SYSTEM AgSYS (* System Configuration *)
  (* Standard: 61499-1 *)
  (* Version 1.0, 2010-04-25, Unknown, TUT *)
  APPLICATION APP1
  END_APPLICATION
  DEVICE HMI : FRAME_DEVICE(BOUNDS := [200,0,800,450], GRID := [3,4])
    RESOURCE HMIPanelMain : PANEL_RESOURCE
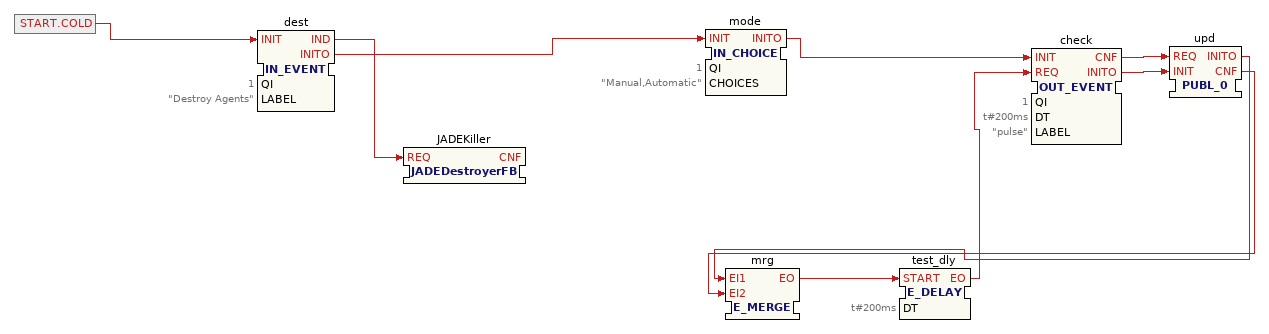
      FBS
        dest : IN_EVENT(QI := 1, LABEL := "Destroy Agents");
        JADEKiller : JADEDestroyerFB;
        mode : IN_CHOICE(QI := 1, CHOICES := "Manual,Automatic");
        check : OUT_EVENT(QI := 1, DT := t#200ms, LABEL := "pulse");
        test_dly : E_DELAY(DT := t#200ms);
        upd : PUBL_0;
        mrg : E_MERGE;
      END_FBS
      EVENT_CONNECTIONS
        START.COLD TO dest.INIT;
        dest.IND TO JADEKiller.REQ;
        dest.INITO TO mode.INIT;
        mode.INITO TO check.INIT;
        test_dly.EO TO check.REQ;
        check.CNF TO upd.REQ;
        upd.INITO TO mrg.EI1;
        upd.CNF TO mrg.EI2;
        mrg.EO TO test_dly.START;
        check.INITO TO upd.INIT;
      END_CONNECTIONS
    END_RESOURCE
    RESOURCE WS2 : PANEL_RESOURCE(ROWS := 4, COLS := 2)
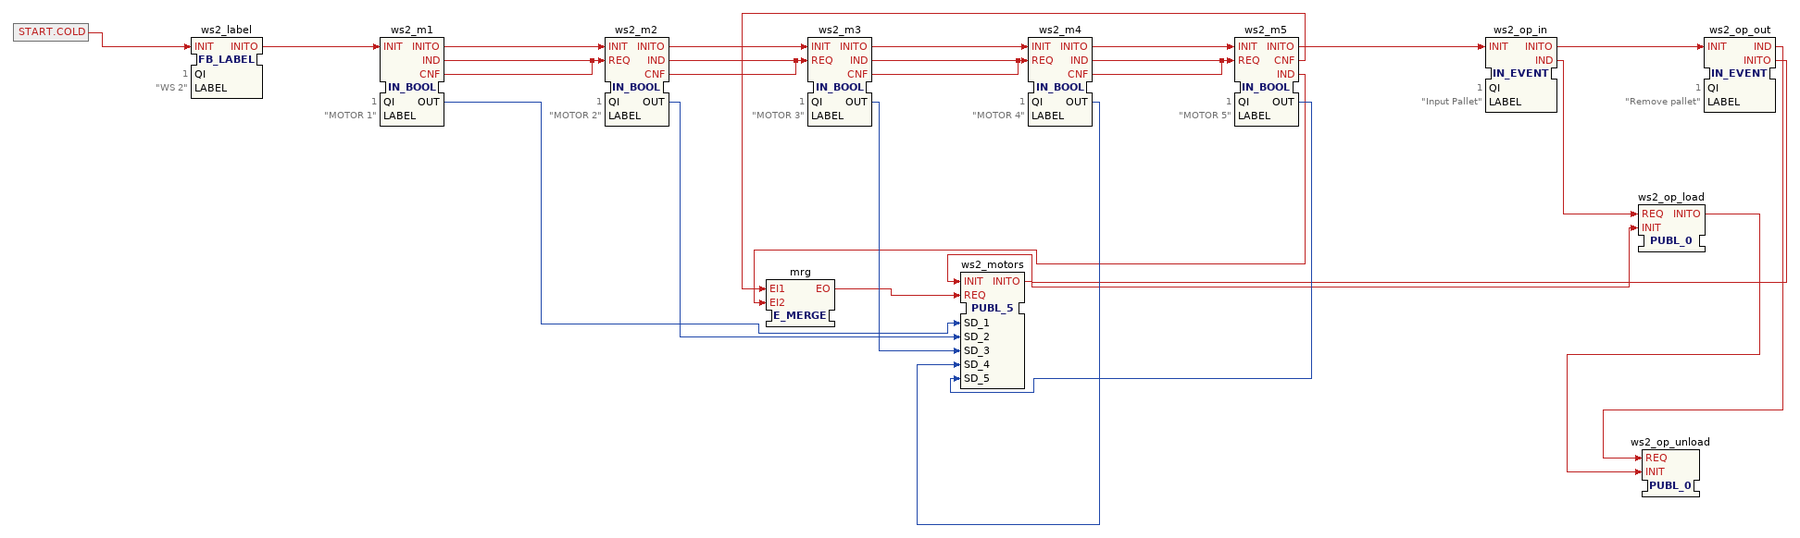
      FBS
        ws2_label : FB_LABEL(QI := 1, LABEL := "WS 2");
        ws2_m1 : IN_BOOL(QI := 1, LABEL := "MOTOR 1");
        ws2_m2 : IN_BOOL(QI := 1, LABEL := "MOTOR 2");
        ws2_m3 : IN_BOOL(QI := 1, LABEL := "MOTOR 3");
        ws2_m4 : IN_BOOL(QI := 1, LABEL := "MOTOR 4");
        ws2_m5 : IN_BOOL(QI := 1, LABEL := "MOTOR 5");
        ws2_op_in : IN_EVENT(QI := 1, LABEL := "Input Pallet");
        ws2_op_out : IN_EVENT(QI := 1, LABEL := "Remove pallet");
        ws2_motors : PUBL_5;
        ws2_op_load : PUBL_0;
        ws2_op_unload : PUBL_0;
        mrg : E_MERGE;
      END_FBS
      EVENT_CONNECTIONS
        START.COLD TO ws2_label.INIT;
        ws2_label.INITO TO ws2_m1.INIT;
        ws2_m1.INITO TO ws2_m2.INIT;
        ws2_m2.INITO TO ws2_m3.INIT;
        ws2_m3.INITO TO ws2_m4.INIT;
        ws2_m4.INITO TO ws2_m5.INIT;
        ws2_m5.INITO TO ws2_op_in.INIT;
        ws2_op_in.INITO TO ws2_op_out.INIT;
        ws2_m1.IND TO ws2_m2.REQ;
        ws2_m2.IND TO ws2_m3.REQ;
        ws2_m3.IND TO ws2_m4.REQ;
        ws2_m4.IND TO ws2_m5.REQ;
        ws2_op_in.IND TO ws2_op_load.REQ;
        ws2_op_out.IND TO ws2_op_unload.REQ;
        ws2_op_out.INITO TO ws2_motors.INIT;
        ws2_motors.INITO TO ws2_op_load.INIT;
        ws2_op_load.INITO TO ws2_op_unload.INIT;
        ws2_m5.CNF TO mrg.EI1;
        ws2_m5.IND TO mrg.EI2;
        mrg.EO TO ws2_motors.REQ;
        ws2_m3.CNF TO ws2_m4.REQ;
        ws2_m4.CNF TO ws2_m5.REQ;
        ws2_m2.CNF TO ws2_m3.REQ;
        ws2_m1.CNF TO ws2_m2.REQ;
      END_CONNECTIONS
      DATA_CONNECTIONS
        ws2_m1.OUT TO ws2_motors.SD_1;
        ws2_m2.OUT TO ws2_motors.SD_2;
        ws2_m3.OUT TO ws2_motors.SD_3;
        ws2_m4.OUT TO ws2_motors.SD_4;
        ws2_m5.OUT TO ws2_motors.SD_5;
      END_CONNECTIONS
    END_RESOURCE
    RESOURCE WS4 : PANEL_RESOURCE(ROWS := 4, COLS := 2)
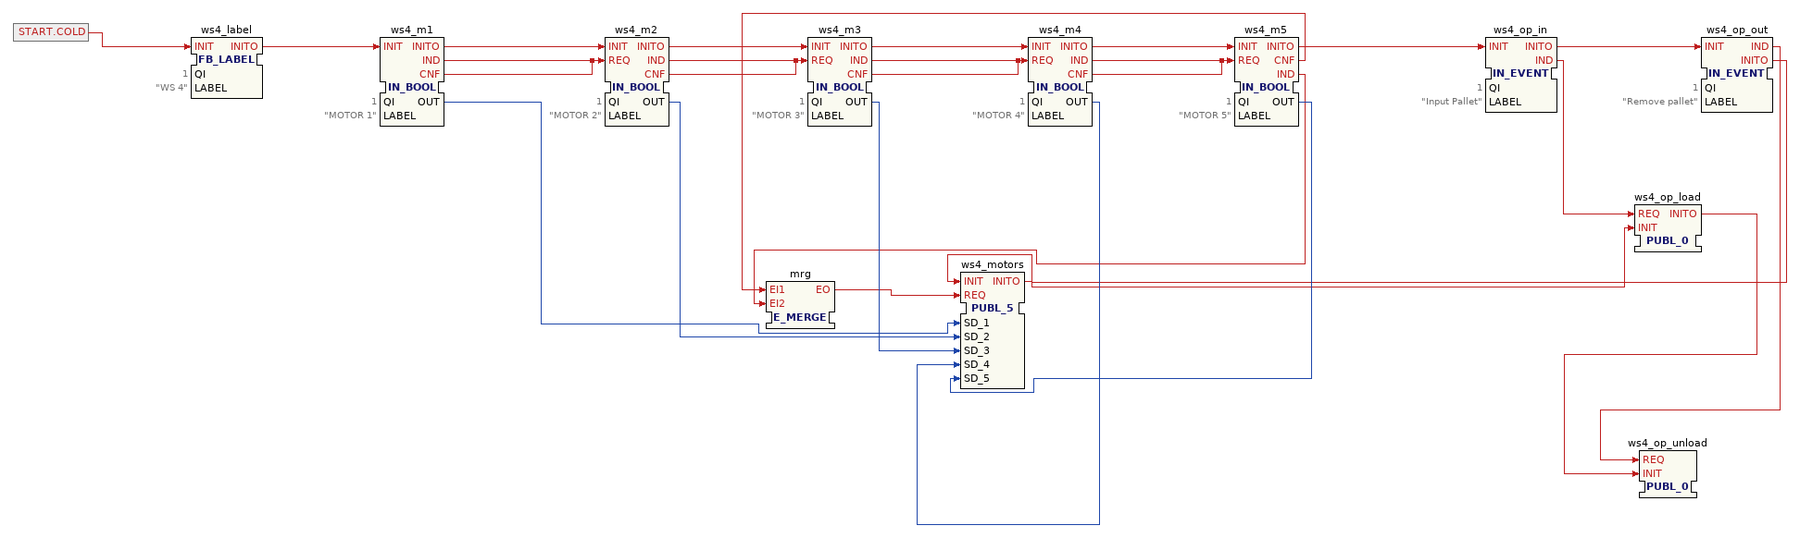
      FBS
        ws4_label : FB_LABEL(QI := 1, LABEL := "WS 4");
        ws4_m1 : IN_BOOL(QI := 1, LABEL := "MOTOR 1");
        ws4_m2 : IN_BOOL(QI := 1, LABEL := "MOTOR 2");
        ws4_m3 : IN_BOOL(QI := 1, LABEL := "MOTOR 3");
        ws4_m4 : IN_BOOL(QI := 1, LABEL := "MOTOR 4");
        ws4_m5 : IN_BOOL(QI := 1, LABEL := "MOTOR 5");
        ws4_op_in : IN_EVENT(QI := 1, LABEL := "Input Pallet");
        ws4_op_out : IN_EVENT(QI := 1, LABEL := "Remove pallet");
        ws4_motors : PUBL_5;
        ws4_op_load : PUBL_0;
        ws4_op_unload : PUBL_0;
        mrg : E_MERGE;
      END_FBS
      EVENT_CONNECTIONS
        START.COLD TO ws4_label.INIT;
        ws4_label.INITO TO ws4_m1.INIT;
        ws4_m1.INITO TO ws4_m2.INIT;
        ws4_m2.INITO TO ws4_m3.INIT;
        ws4_m3.INITO TO ws4_m4.INIT;
        ws4_m4.INITO TO ws4_m5.INIT;
        ws4_m5.INITO TO ws4_op_in.INIT;
        ws4_op_in.INITO TO ws4_op_out.INIT;
        ws4_m1.IND TO ws4_m2.REQ;
        ws4_m2.IND TO ws4_m3.REQ;
        ws4_m3.IND TO ws4_m4.REQ;
        ws4_m4.IND TO ws4_m5.REQ;
        ws4_op_in.IND TO ws4_op_load.REQ;
        ws4_op_out.IND TO ws4_op_unload.REQ;
        ws4_op_out.INITO TO ws4_motors.INIT;
        ws4_motors.INITO TO ws4_op_load.INIT;
        ws4_op_load.INITO TO ws4_op_unload.INIT;
        ws4_m5.CNF TO mrg.EI1;
        ws4_m5.IND TO mrg.EI2;
        mrg.EO TO ws4_motors.REQ;
        ws4_m3.CNF TO ws4_m4.REQ;
        ws4_m4.CNF TO ws4_m5.REQ;
        ws4_m2.CNF TO ws4_m3.REQ;
        ws4_m1.CNF TO ws4_m2.REQ;
      END_CONNECTIONS
      DATA_CONNECTIONS
        ws4_m1.OUT TO ws4_motors.SD_1;
        ws4_m2.OUT TO ws4_motors.SD_2;
        ws4_m3.OUT TO ws4_motors.SD_3;
        ws4_m4.OUT TO ws4_motors.SD_4;
        ws4_m5.OUT TO ws4_motors.SD_5;
      END_CONNECTIONS
    END_RESOURCE
    RESOURCE empt1 : PANEL_RESOURCE
    END_RESOURCE
    RESOURCE Start_Lifter : PANEL_RESOURCE(ROWS := 3, COLS := 1)
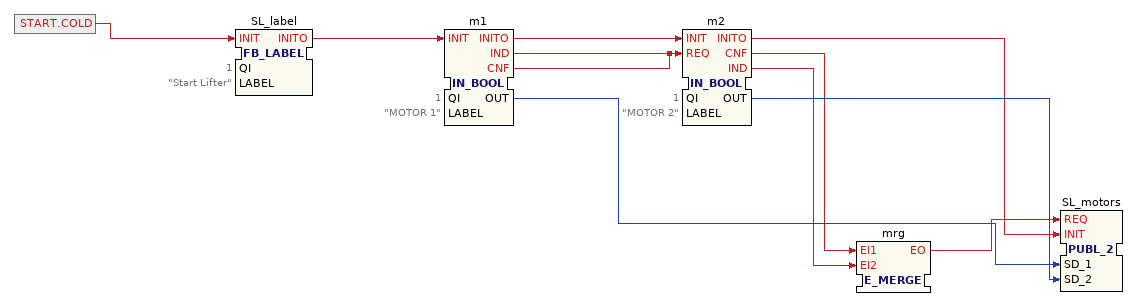
      FBS
        SL_label : FB_LABEL(QI := 1, LABEL := "Start Lifter");
        m1 : IN_BOOL(QI := 1, LABEL := "MOTOR 1");
        m2 : IN_BOOL(QI := 1, LABEL := "MOTOR 2");
        SL_motors : PUBL_2;
        mrg : E_MERGE;
      END_FBS
      EVENT_CONNECTIONS
        START.COLD TO SL_label.INIT;
        m1.INITO TO m2.INIT;
        m1.IND TO m2.REQ;
        mrg.EO TO SL_motors.REQ;
        m1.CNF TO m2.REQ;
        m2.INITO TO SL_motors.INIT;
        m2.CNF TO mrg.EI1;
        m2.IND TO mrg.EI2;
        SL_label.INITO TO m1.INIT;
      END_CONNECTIONS
      DATA_CONNECTIONS
        m1.OUT TO SL_motors.SD_1;
        m2.OUT TO SL_motors.SD_2;
      END_CONNECTIONS
    END_RESOURCE
    RESOURCE ML1 : PANEL_RESOURCE(ROWS := 3, COLS := 2)
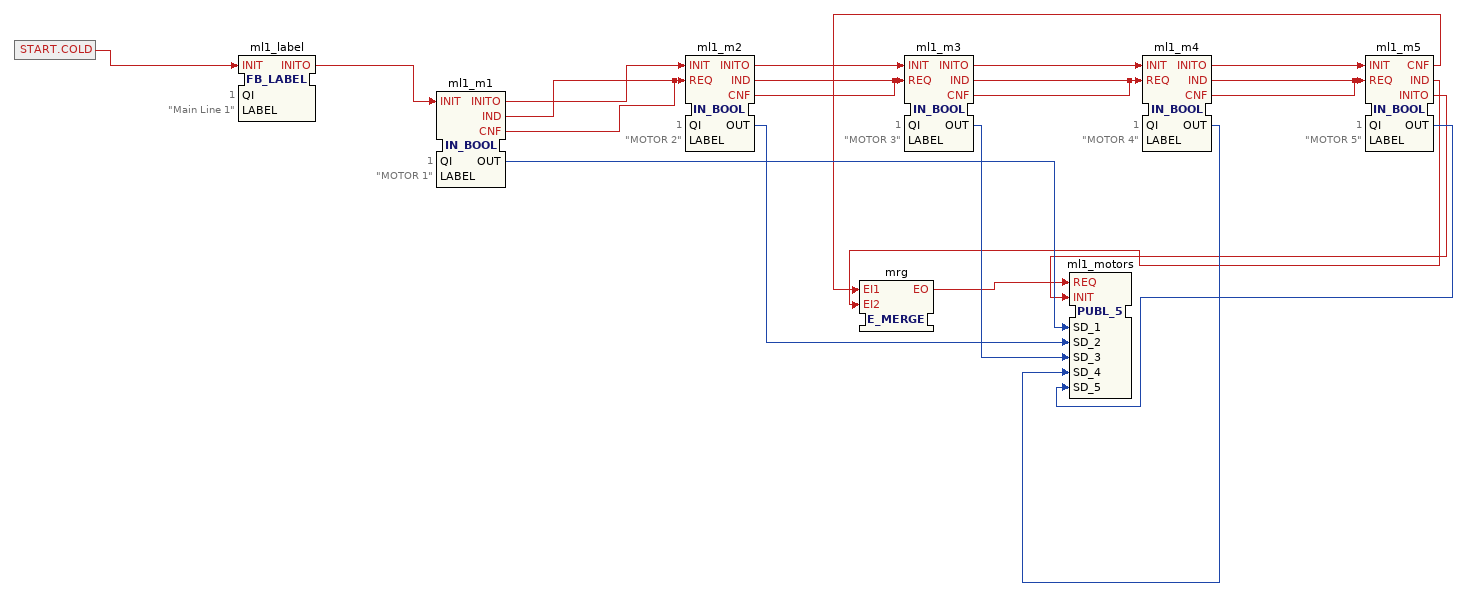
      FBS
        ml1_label : FB_LABEL(QI := 1, LABEL := "Main Line 1");
        ml1_m1 : IN_BOOL(QI := 1, LABEL := "MOTOR 1");
        ml1_m2 : IN_BOOL(QI := 1, LABEL := "MOTOR 2");
        ml1_m3 : IN_BOOL(QI := 1, LABEL := "MOTOR 3");
        ml1_m4 : IN_BOOL(QI := 1, LABEL := "MOTOR 4");
        ml1_m5 : IN_BOOL(QI := 1, LABEL := "MOTOR 5");
        ml1_motors : PUBL_5;
        mrg : E_MERGE;
      END_FBS
      EVENT_CONNECTIONS
        START.COLD TO ml1_label.INIT;
        ml1_m1.INITO TO ml1_m2.INIT;
        ml1_m2.INITO TO ml1_m3.INIT;
        ml1_m3.INITO TO ml1_m4.INIT;
        ml1_m4.INITO TO ml1_m5.INIT;
        ml1_m1.IND TO ml1_m2.REQ;
        ml1_m2.IND TO ml1_m3.REQ;
        ml1_m3.IND TO ml1_m4.REQ;
        ml1_m4.IND TO ml1_m5.REQ;
        ml1_m5.CNF TO mrg.EI1;
        ml1_m5.IND TO mrg.EI2;
        mrg.EO TO ml1_motors.REQ;
        ml1_m3.CNF TO ml1_m4.REQ;
        ml1_m4.CNF TO ml1_m5.REQ;
        ml1_m2.CNF TO ml1_m3.REQ;
        ml1_m1.CNF TO ml1_m2.REQ;
        ml1_m5.INITO TO ml1_motors.INIT;
        ml1_label.INITO TO ml1_m1.INIT;
      END_CONNECTIONS
      DATA_CONNECTIONS
        ml1_m1.OUT TO ml1_motors.SD_1;
        ml1_m2.OUT TO ml1_motors.SD_2;
        ml1_m3.OUT TO ml1_motors.SD_3;
        ml1_m4.OUT TO ml1_motors.SD_4;
        ml1_m5.OUT TO ml1_motors.SD_5;
      END_CONNECTIONS
    END_RESOURCE
    RESOURCE ML2 : PANEL_RESOURCE(ROWS := 3, COLS := 2)
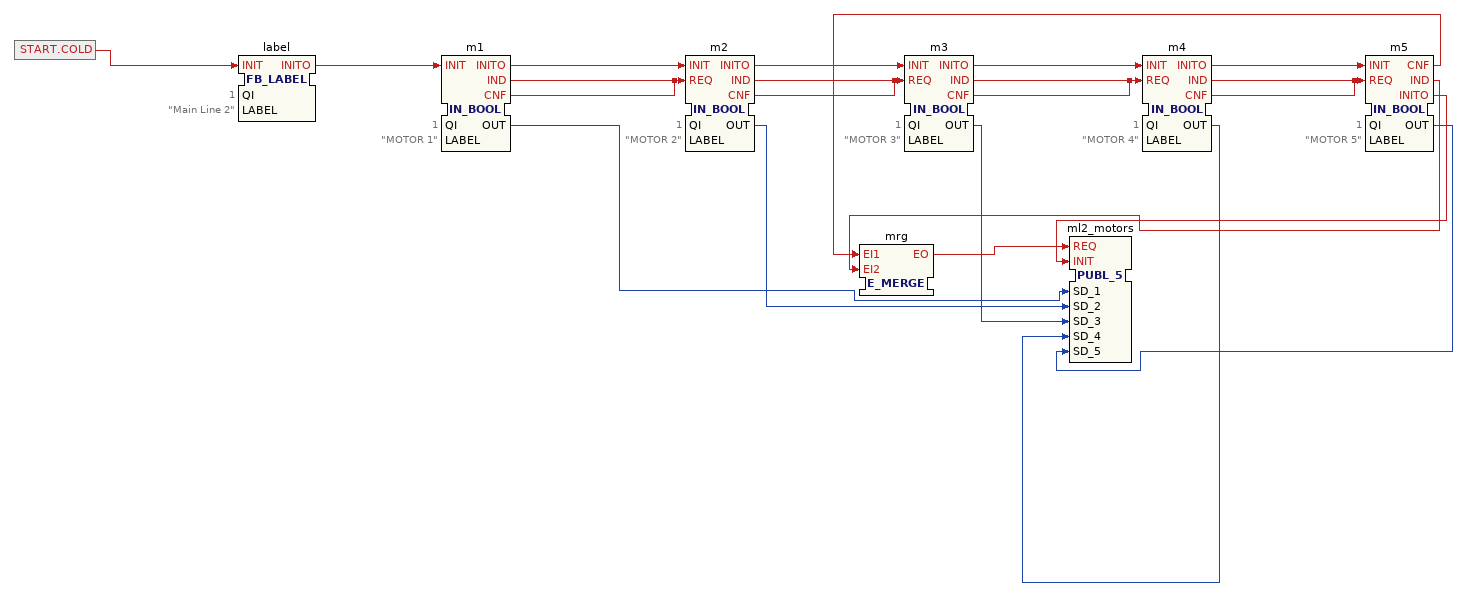
      FBS
        label : FB_LABEL(QI := 1, LABEL := "Main Line 2");
        m1 : IN_BOOL(QI := 1, LABEL := "MOTOR 1");
        m2 : IN_BOOL(QI := 1, LABEL := "MOTOR 2");
        m3 : IN_BOOL(QI := 1, LABEL := "MOTOR 3");
        m4 : IN_BOOL(QI := 1, LABEL := "MOTOR 4");
        m5 : IN_BOOL(QI := 1, LABEL := "MOTOR 5");
        ml2_motors : PUBL_5;
        mrg : E_MERGE;
      END_FBS
      EVENT_CONNECTIONS
        START.COLD TO label.INIT;
        m1.INITO TO m2.INIT;
        m2.INITO TO m3.INIT;
        m3.INITO TO m4.INIT;
        m4.INITO TO m5.INIT;
        m1.IND TO m2.REQ;
        m2.IND TO m3.REQ;
        m3.IND TO m4.REQ;
        m4.IND TO m5.REQ;
        m5.CNF TO mrg.EI1;
        m5.IND TO mrg.EI2;
        mrg.EO TO ml2_motors.REQ;
        m3.CNF TO m4.REQ;
        m4.CNF TO m5.REQ;
        m2.CNF TO m3.REQ;
        m1.CNF TO m2.REQ;
        m5.INITO TO ml2_motors.INIT;
        label.INITO TO m1.INIT;
      END_CONNECTIONS
      DATA_CONNECTIONS
        m1.OUT TO ml2_motors.SD_1;
        m2.OUT TO ml2_motors.SD_2;
        m3.OUT TO ml2_motors.SD_3;
        m4.OUT TO ml2_motors.SD_4;
        m5.OUT TO ml2_motors.SD_5;
      END_CONNECTIONS
    END_RESOURCE
    RESOURCE End_Lifter : PANEL_RESOURCE(ROWS := 3, COLS := 1)
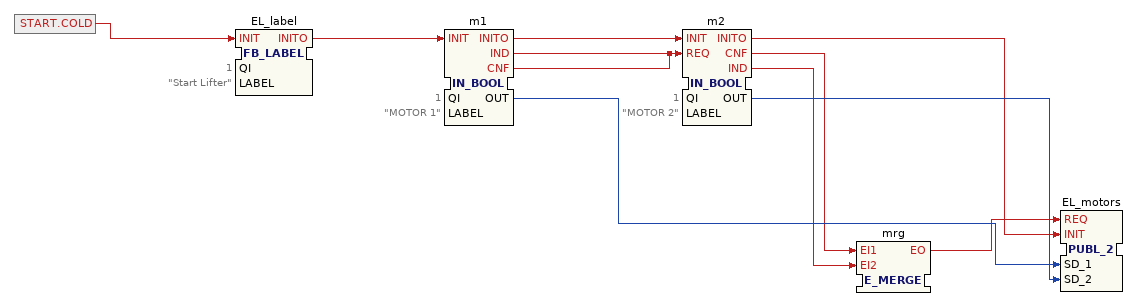
      FBS
        EL_label : FB_LABEL(QI := 1, LABEL := "Start Lifter");
        m1 : IN_BOOL(QI := 1, LABEL := "MOTOR 1");
        m2 : IN_BOOL(QI := 1, LABEL := "MOTOR 2");
        EL_motors : PUBL_2;
        mrg : E_MERGE;
      END_FBS
      EVENT_CONNECTIONS
        START.COLD TO EL_label.INIT;
        m1.INITO TO m2.INIT;
        m1.IND TO m2.REQ;
        mrg.EO TO EL_motors.REQ;
        m1.CNF TO m2.REQ;
        m2.INITO TO EL_motors.INIT;
        m2.CNF TO mrg.EI1;
        m2.IND TO mrg.EI2;
        EL_label.INITO TO m1.INIT;
      END_CONNECTIONS
      DATA_CONNECTIONS
        m1.OUT TO EL_motors.SD_1;
        m2.OUT TO EL_motors.SD_2;
      END_CONNECTIONS
    END_RESOURCE
    RESOURCE empt2 : PANEL_RESOURCE
    END_RESOURCE
    RESOURCE WS1 : PANEL_RESOURCE(ROWS := 4, COLS := 2)
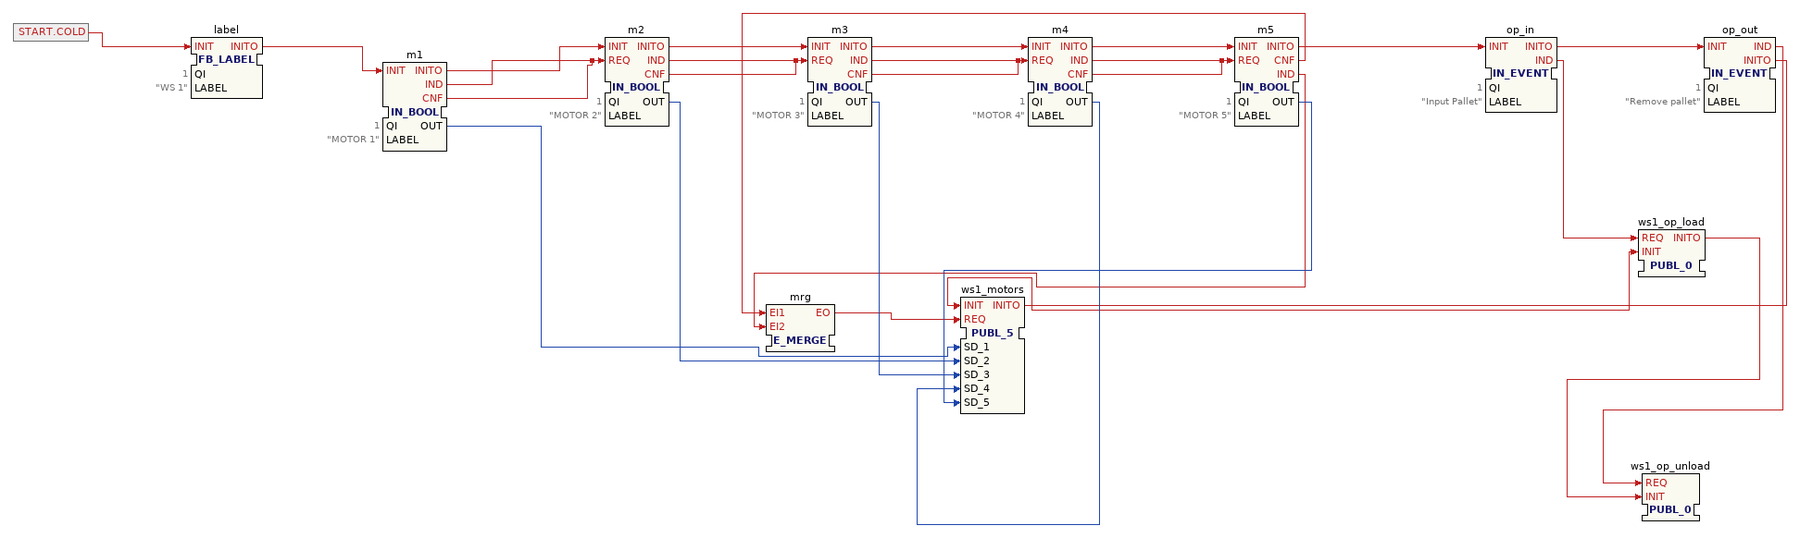
      FBS
        label : FB_LABEL(QI := 1, LABEL := "WS 1");
        m1 : IN_BOOL(QI := 1, LABEL := "MOTOR 1");
        m2 : IN_BOOL(QI := 1, LABEL := "MOTOR 2");
        m3 : IN_BOOL(QI := 1, LABEL := "MOTOR 3");
        m4 : IN_BOOL(QI := 1, LABEL := "MOTOR 4");
        m5 : IN_BOOL(QI := 1, LABEL := "MOTOR 5");
        op_in : IN_EVENT(QI := 1, LABEL := "Input Pallet");
        op_out : IN_EVENT(QI := 1, LABEL := "Remove pallet");
        ws1_motors : PUBL_5;
        ws1_op_load : PUBL_0;
        ws1_op_unload : PUBL_0;
        mrg : E_MERGE;
      END_FBS
      EVENT_CONNECTIONS
        START.COLD TO label.INIT;
        m1.INITO TO m2.INIT;
        m2.INITO TO m3.INIT;
        m3.INITO TO m4.INIT;
        m4.INITO TO m5.INIT;
        m5.INITO TO op_in.INIT;
        op_in.INITO TO op_out.INIT;
        m1.IND TO m2.REQ;
        m2.IND TO m3.REQ;
        m3.IND TO m4.REQ;
        m4.IND TO m5.REQ;
        op_in.IND TO ws1_op_load.REQ;
        op_out.IND TO ws1_op_unload.REQ;
        op_out.INITO TO ws1_motors.INIT;
        ws1_motors.INITO TO ws1_op_load.INIT;
        ws1_op_load.INITO TO ws1_op_unload.INIT;
        m5.CNF TO mrg.EI1;
        m5.IND TO mrg.EI2;
        mrg.EO TO ws1_motors.REQ;
        m3.CNF TO m4.REQ;
        m4.CNF TO m5.REQ;
        m2.CNF TO m3.REQ;
        m1.CNF TO m2.REQ;
        label.INITO TO m1.INIT;
      END_CONNECTIONS
      DATA_CONNECTIONS
        m1.OUT TO ws1_motors.SD_1;
        m2.OUT TO ws1_motors.SD_2;
        m3.OUT TO ws1_motors.SD_3;
        m4.OUT TO ws1_motors.SD_4;
        m5.OUT TO ws1_motors.SD_5;
      END_CONNECTIONS
    END_RESOURCE
    RESOURCE WS3 : PANEL_RESOURCE(ROWS := 4, COLS := 2)
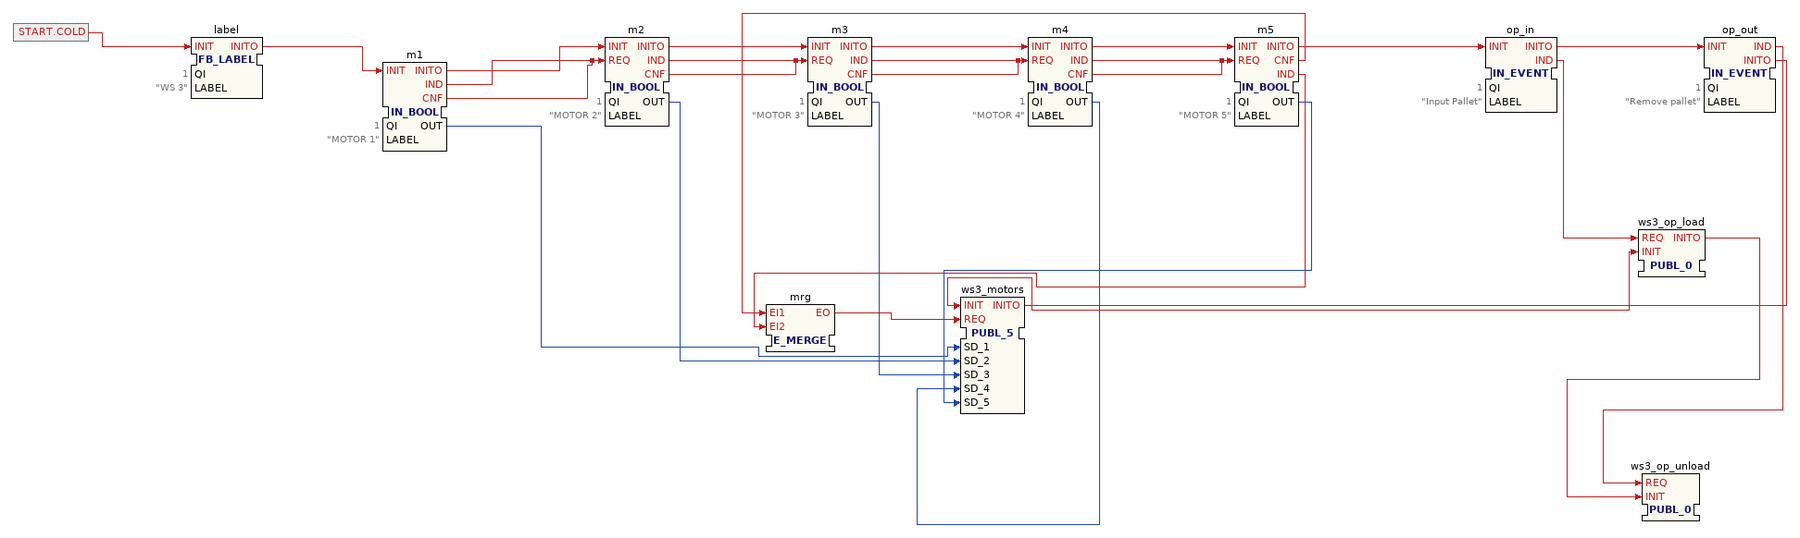
      FBS
        label : FB_LABEL(QI := 1, LABEL := "WS 3");
        m1 : IN_BOOL(QI := 1, LABEL := "MOTOR 1");
        m2 : IN_BOOL(QI := 1, LABEL := "MOTOR 2");
        m3 : IN_BOOL(QI := 1, LABEL := "MOTOR 3");
        m4 : IN_BOOL(QI := 1, LABEL := "MOTOR 4");
        m5 : IN_BOOL(QI := 1, LABEL := "MOTOR 5");
        op_in : IN_EVENT(QI := 1, LABEL := "Input Pallet");
        op_out : IN_EVENT(QI := 1, LABEL := "Remove pallet");
        ws3_motors : PUBL_5;
        ws3_op_load : PUBL_0;
        ws3_op_unload : PUBL_0;
        mrg : E_MERGE;
      END_FBS
      EVENT_CONNECTIONS
        START.COLD TO label.INIT;
        m1.INITO TO m2.INIT;
        m2.INITO TO m3.INIT;
        m3.INITO TO m4.INIT;
        m4.INITO TO m5.INIT;
        m5.INITO TO op_in.INIT;
        op_in.INITO TO op_out.INIT;
        m1.IND TO m2.REQ;
        m2.IND TO m3.REQ;
        m3.IND TO m4.REQ;
        m4.IND TO m5.REQ;
        op_in.IND TO ws3_op_load.REQ;
        op_out.IND TO ws3_op_unload.REQ;
        op_out.INITO TO ws3_motors.INIT;
        ws3_motors.INITO TO ws3_op_load.INIT;
        ws3_op_load.INITO TO ws3_op_unload.INIT;
        m5.CNF TO mrg.EI1;
        m5.IND TO mrg.EI2;
        mrg.EO TO ws3_motors.REQ;
        m3.CNF TO m4.REQ;
        m4.CNF TO m5.REQ;
        m2.CNF TO m3.REQ;
        m1.CNF TO m2.REQ;
        label.INITO TO m1.INIT;
      END_CONNECTIONS
      DATA_CONNECTIONS
        m1.OUT TO ws3_motors.SD_1;
        m2.OUT TO ws3_motors.SD_2;
        m3.OUT TO ws3_motors.SD_3;
        m4.OUT TO ws3_motors.SD_4;
        m5.OUT TO ws3_motors.SD_5;
      END_CONNECTIONS
    END_RESOURCE
    RESOURCE empt3 : PANEL_RESOURCE
    END_RESOURCE
  END_DEVICE
  DEVICE Control : FRAME_DEVICE
    RESOURCE ControlContainer : PANEL_RESOURCE
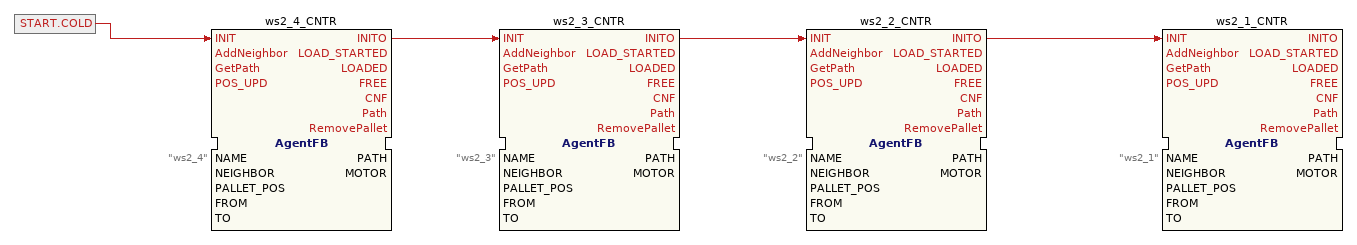
      FBS
        ws2_4_CNTR : AgentFB(NAME := "ws2_4");
        ws2_3_CNTR : AgentFB(NAME := "ws2_3");
        ws2_2_CNTR : AgentFB(NAME := "ws2_2");
        ws2_1_CNTR : AgentFB(NAME := "ws2_1");
      END_FBS
      EVENT_CONNECTIONS
        START.COLD TO ws2_4_CNTR.INIT;
        ws2_4_CNTR.INITO TO ws2_3_CNTR.INIT;
        ws2_3_CNTR.INITO TO ws2_2_CNTR.INIT;
        ws2_2_CNTR.INITO TO ws2_1_CNTR.INIT;
      END_CONNECTIONS
    END_RESOURCE
  END_DEVICE
  DEVICE Model : FRAME_DEVICE
    RESOURCE WS2_model : PANEL_RESOURCE
      FBS
        ws2_1 : CNV_MDL(WKPC := [255,255,0], STYLE := VSTYLE#PALLET, VF := 10);
        ws2_2 : CNV_MDL(WKPC := [255,255,0], STYLE := VSTYLE#PALLET, VF := 10);
        ws2_3 : CNV_MDL(VF := 10, STYLE := VSTYLE#PALLET, WKPC := [255,255,0]);
        ws2_4 : CNV_MDL(VF := 10, STYLE := VSTYLE#PALLET, WKPC := [255,255,0]);
        ws2_5 : CNV_MDL(WKPC := [255,255,0], STYLE := VSTYLE#PALLET, VF := 10);
        ws2_pos : PUBL_5;
        ws2_sty : PUBL_5;
        ws2_motors : SUBL_5;
        ws2_op_load : SUBL_0;
        ws2_op_unload : SUBL_0;
        split5 : E_SPLIT;
        split4 : E_SPLIT;
        split3 : E_SPLIT;
        split2 : E_SPLIT;
        split1 : E_SPLIT;
        upd : SUBL_0;
        sync_prev_1 : ConvSync(STYLE1 := VSTYLE#NONE);
        sync1_2 : ConvSync(STYLE1 := VSTYLE#NONE);
        sync2_3 : ConvSync(STYLE1 := VSTYLE#NONE);
        sync4_5 : ConvSync(STYLE1 := VSTYLE#NONE);
        sync3_4 : ConvSync(STYLE1 := VSTYLE#NONE);
        ml1_out1 : SUBL_2;
        ws2_in : PUBL_0;
        ml1_in1 : SUBL_0;
        ws2_out : PUBL_2;
      END_FBS
      EVENT_CONNECTIONS
        START.COLD TO ws2_motors.INIT;
        ws2_motors.INITO TO ws2_pos.INIT;
        ws2_pos.INITO TO ws2_sty.INIT;
        ws2_sty.INITO TO ws2_op_load.INIT;
        ws2_op_load.INITO TO ws2_op_unload.INIT;
        ws2_op_load.IND TO ws2_3.LOAD;
        ws2_op_unload.IND TO ws2_3.UNLD;
        ws2_pos.CNF TO ws2_sty.REQ;
        split1.EO2 TO split2.EI;
        split1.EO1 TO ws2_1.CLK;
        split2.EO2 TO split3.EI;
        split2.EO1 TO ws2_2.CLK;
        split3.EO2 TO split4.EI;
        split3.EO1 TO ws2_3.CLK;
        split4.EO2 TO split5.EI;
        split4.EO1 TO ws2_5.CLK;
        ws2_op_unload.INITO TO upd.INIT;
        upd.IND TO split1.EI;
        split5.EO2 TO ws2_pos.REQ;
        split5.EO1 TO ws2_4.CLK;
        sync3_4.CNF TO ws2_3.UNLD;
        sync3_4.CNF TO ws2_4.LOAD;
        split4.EO1 TO sync4_5.REQ;
        sync4_5.CNF TO ws2_4.UNLD;
        sync4_5.CNF TO ws2_5.LOAD;
        split3.EO1 TO sync3_4.REQ;
        split1.EO1 TO sync1_2.REQ;
        sync1_2.CNF TO ws2_2.LOAD;
        sync1_2.CNF TO ws2_1.UNLD;
        split2.EO1 TO sync2_3.REQ;
        upd.INITO TO ml1_out1.INIT;
        ml1_out1.IND TO sync_prev_1.REQ;
        sync_prev_1.CNF TO ws2_in.REQ;
        ml1_out1.INITO TO ws2_in.INIT;
        sync_prev_1.CNF TO ws2_1.LOAD;
        ws2_op_unload.INITO TO ml1_in1.INIT;
        ml1_in1.IND TO ws2_5.UNLD;
        ml1_in1.INITO TO ws2_out.INIT;
        ws2_sty.CNF TO ws2_out.REQ;
        sync2_3.CNF TO ws2_3.LOAD;
        sync2_3.CNF TO ws2_2.UNLD;
      END_CONNECTIONS
      DATA_CONNECTIONS
        ws2_1.POS TO ws2_pos.SD_1;
        ws2_2.POS TO ws2_pos.SD_2;
        ws2_3.POS TO ws2_pos.SD_3;
        ws2_4.POS TO ws2_pos.SD_4;
        ws2_5.POS TO ws2_pos.SD_5;
        ws2_1.STYLO TO ws2_sty.SD_1;
        ws2_2.STYLO TO ws2_sty.SD_2;
        ws2_3.STYLO TO ws2_sty.SD_3;
        ws2_4.STYLO TO ws2_sty.SD_4;
        ws2_5.STYLO TO ws2_sty.SD_5;
        ws2_motors.RD_2 TO ws2_2.MTR_ON;
        ws2_motors.RD_3 TO ws2_3.MTR_ON;
        ws2_motors.RD_4 TO ws2_4.MTR_ON;
        ws2_motors.RD_5 TO ws2_5.MTR_ON;
        ws2_3.END TO sync3_4.END1;
        ws2_motors.RD_3 TO sync3_4.MOTOR1;
        ws2_motors.RD_4 TO sync3_4.MOTOR2;
        ws2_4.STYLO TO sync3_4.STYLE2;
        ws2_motors.RD_1 TO ws2_1.MTR_ON;
        ws2_4.END TO sync4_5.END1;
        ws2_motors.RD_4 TO sync4_5.MOTOR1;
        ws2_motors.RD_5 TO sync4_5.MOTOR2;
        ws2_5.STYLO TO sync4_5.STYLE2;
        ws2_1.END TO sync1_2.END1;
        ws2_motors.RD_1 TO sync1_2.MOTOR1;
        ws2_motors.RD_2 TO sync1_2.MOTOR2;
        ws2_2.STYLO TO sync1_2.STYLE2;
        ws2_motors.RD_2 TO sync2_3.MOTOR1;
        ws2_motors.RD_3 TO sync2_3.MOTOR2;
        ws2_3.STYLO TO sync2_3.STYLE2;
        ws2_2.END TO sync2_3.END1;
        ws2_motors.RD_1 TO sync_prev_1.MOTOR1;
        ws2_5.END TO ws2_out.SD_1;
        ws2_motors.RD_5 TO ws2_out.SD_2;
        ml1_out1.RD_1 TO sync_prev_1.END1;
        ml1_out1.RD_2 TO sync_prev_1.MOTOR2;
        ws2_1.STYLO TO sync_prev_1.STYLE2;
      END_CONNECTIONS
    END_RESOURCE
    RESOURCE WS4_model : PANEL_RESOURCE
      FBS
        ws4_1 : CNV_MDL(WKPC := [255,255,0], STYLE := VSTYLE#PALLET, VF := 10);
        ws4_2 : CNV_MDL(WKPC := [255,255,0], STYLE := VSTYLE#PALLET, VF := 10);
        ws4_3 : CNV_MDL(VF := 10, STYLE := VSTYLE#PALLET, WKPC := [255,255,0]);
        ws4_4 : CNV_MDL(VF := 10, STYLE := VSTYLE#PALLET, WKPC := [255,255,0]);
        ws4_5 : CNV_MDL(WKPC := [255,255,0], STYLE := VSTYLE#PALLET, VF := 10);
        ws4_pos : PUBL_5;
        ws4_sty : PUBL_5;
        ws4_motors : SUBL_5;
        ws4_op_load : SUBL_0;
        ws4_op_unload : SUBL_0;
        split5 : E_SPLIT;
        split4 : E_SPLIT;
        split3 : E_SPLIT;
        split2 : E_SPLIT;
        split1 : E_SPLIT;
        upd : SUBL_0;
        sync1_2 : ConvSync(STYLE1 := VSTYLE#NONE);
        sync2_3 : ConvSync(STYLE1 := VSTYLE#NONE);
        sync4_5 : ConvSync(STYLE1 := VSTYLE#NONE);
        sync3_4 : ConvSync(STYLE1 := VSTYLE#NONE);
      END_FBS
      EVENT_CONNECTIONS
        START.COLD TO ws4_motors.INIT;
        ws4_motors.INITO TO ws4_pos.INIT;
        ws4_pos.INITO TO ws4_sty.INIT;
        ws4_sty.INITO TO ws4_op_load.INIT;
        ws4_op_load.INITO TO ws4_op_unload.INIT;
        ws4_op_load.IND TO ws4_3.LOAD;
        ws4_op_unload.IND TO ws4_3.UNLD;
        ws4_pos.CNF TO ws4_sty.REQ;
        split1.EO2 TO split2.EI;
        split1.EO1 TO ws4_1.CLK;
        split2.EO2 TO split3.EI;
        split2.EO1 TO ws4_2.CLK;
        split3.EO2 TO split4.EI;
        split3.EO1 TO ws4_3.CLK;
        split4.EO2 TO split5.EI;
        split4.EO1 TO ws4_5.CLK;
        ws4_op_unload.INITO TO upd.INIT;
        upd.IND TO split1.EI;
        split5.EO2 TO ws4_pos.REQ;
        split5.EO1 TO ws4_4.CLK;
        sync3_4.CNF TO ws4_3.UNLD;
        sync3_4.CNF TO ws4_4.LOAD;
        split4.EO1 TO sync4_5.REQ;
        sync4_5.CNF TO ws4_4.UNLD;
        sync4_5.CNF TO ws4_5.LOAD;
        split3.EO1 TO sync3_4.REQ;
        split1.EO1 TO sync1_2.REQ;
        sync1_2.CNF TO ws4_2.LOAD;
        sync1_2.CNF TO ws4_1.UNLD;
        split2.EO1 TO sync2_3.REQ;
        sync2_3.CNF TO ws4_3.LOAD;
        sync2_3.CNF TO ws4_2.UNLD;
      END_CONNECTIONS
      DATA_CONNECTIONS
        ws4_1.POS TO ws4_pos.SD_1;
        ws4_2.POS TO ws4_pos.SD_2;
        ws4_3.POS TO ws4_pos.SD_3;
        ws4_4.POS TO ws4_pos.SD_4;
        ws4_5.POS TO ws4_pos.SD_5;
        ws4_1.STYLO TO ws4_sty.SD_1;
        ws4_2.STYLO TO ws4_sty.SD_2;
        ws4_3.STYLO TO ws4_sty.SD_3;
        ws4_4.STYLO TO ws4_sty.SD_4;
        ws4_5.STYLO TO ws4_sty.SD_5;
        ws4_motors.RD_2 TO ws4_2.MTR_ON;
        ws4_motors.RD_3 TO ws4_3.MTR_ON;
        ws4_motors.RD_4 TO ws4_4.MTR_ON;
        ws4_motors.RD_5 TO ws4_5.MTR_ON;
        ws4_3.END TO sync3_4.END1;
        ws4_motors.RD_3 TO sync3_4.MOTOR1;
        ws4_motors.RD_4 TO sync3_4.MOTOR2;
        ws4_4.STYLO TO sync3_4.STYLE2;
        ws4_motors.RD_1 TO ws4_1.MTR_ON;
        ws4_4.END TO sync4_5.END1;
        ws4_motors.RD_4 TO sync4_5.MOTOR1;
        ws4_motors.RD_5 TO sync4_5.MOTOR2;
        ws4_5.STYLO TO sync4_5.STYLE2;
        ws4_1.END TO sync1_2.END1;
        ws4_motors.RD_1 TO sync1_2.MOTOR1;
        ws4_motors.RD_2 TO sync1_2.MOTOR2;
        ws4_2.STYLO TO sync1_2.STYLE2;
        ws4_motors.RD_2 TO sync2_3.MOTOR1;
        ws4_motors.RD_3 TO sync2_3.MOTOR2;
        ws4_3.STYLO TO sync2_3.STYLE2;
        ws4_2.END TO sync2_3.END1;
      END_CONNECTIONS
    END_RESOURCE
    RESOURCE WS1_model : PANEL_RESOURCE
      FBS
        ws1_1 : CNV_MDL(WKPC := [255,255,0], STYLE := VSTYLE#PALLET, VF := 10);
        ws1_2 : CNV_MDL(WKPC := [255,255,0], STYLE := VSTYLE#PALLET, VF := 10);
        ws1_3 : CNV_MDL(VF := 10, STYLE := VSTYLE#PALLET, WKPC := [255,255,0]);
        ws1_4 : CNV_MDL(VF := 10, STYLE := VSTYLE#PALLET, WKPC := [255,255,0]);
        ws1_5 : CNV_MDL(WKPC := [255,255,0], STYLE := VSTYLE#PALLET, VF := 10);
        ws1_pos : PUBL_5;
        ws1_sty : PUBL_5;
        ws1_motors : SUBL_5;
        ws1_op_load : SUBL_0;
        ws1_op_unload : SUBL_0;
        split5 : E_SPLIT;
        split4 : E_SPLIT;
        split3 : E_SPLIT;
        split2 : E_SPLIT;
        split1 : E_SPLIT;
        upd : SUBL_0;
        sync1_2 : ConvSync(STYLE1 := VSTYLE#NONE);
        sync2_3 : ConvSync(STYLE1 := VSTYLE#NONE);
        sync4_5 : ConvSync(STYLE1 := VSTYLE#NONE);
        sync3_4 : ConvSync(STYLE1 := VSTYLE#NONE);
      END_FBS
      EVENT_CONNECTIONS
        START.COLD TO ws1_motors.INIT;
        ws1_motors.INITO TO ws1_pos.INIT;
        ws1_pos.INITO TO ws1_sty.INIT;
        ws1_sty.INITO TO ws1_op_load.INIT;
        ws1_op_load.INITO TO ws1_op_unload.INIT;
        ws1_op_load.IND TO ws1_3.LOAD;
        ws1_op_unload.IND TO ws1_3.UNLD;
        ws1_pos.CNF TO ws1_sty.REQ;
        split1.EO2 TO split2.EI;
        split1.EO1 TO ws1_1.CLK;
        split2.EO2 TO split3.EI;
        split2.EO1 TO ws1_2.CLK;
        split3.EO2 TO split4.EI;
        split3.EO1 TO ws1_3.CLK;
        split4.EO2 TO split5.EI;
        split4.EO1 TO ws1_5.CLK;
        ws1_op_unload.INITO TO upd.INIT;
        upd.IND TO split1.EI;
        split5.EO2 TO ws1_pos.REQ;
        split5.EO1 TO ws1_4.CLK;
        sync3_4.CNF TO ws1_3.UNLD;
        sync3_4.CNF TO ws1_4.LOAD;
        split4.EO1 TO sync4_5.REQ;
        sync4_5.CNF TO ws1_4.UNLD;
        sync4_5.CNF TO ws1_5.LOAD;
        split3.EO1 TO sync3_4.REQ;
        split1.EO1 TO sync1_2.REQ;
        sync1_2.CNF TO ws1_2.LOAD;
        sync1_2.CNF TO ws1_1.UNLD;
        split2.EO1 TO sync2_3.REQ;
        sync2_3.CNF TO ws1_3.LOAD;
        sync2_3.CNF TO ws1_2.UNLD;
      END_CONNECTIONS
      DATA_CONNECTIONS
        ws1_1.POS TO ws1_pos.SD_1;
        ws1_2.POS TO ws1_pos.SD_2;
        ws1_3.POS TO ws1_pos.SD_3;
        ws1_4.POS TO ws1_pos.SD_4;
        ws1_5.POS TO ws1_pos.SD_5;
        ws1_1.STYLO TO ws1_sty.SD_1;
        ws1_2.STYLO TO ws1_sty.SD_2;
        ws1_3.STYLO TO ws1_sty.SD_3;
        ws1_4.STYLO TO ws1_sty.SD_4;
        ws1_5.STYLO TO ws1_sty.SD_5;
        ws1_motors.RD_2 TO ws1_2.MTR_ON;
        ws1_motors.RD_3 TO ws1_3.MTR_ON;
        ws1_motors.RD_4 TO ws1_4.MTR_ON;
        ws1_motors.RD_5 TO ws1_5.MTR_ON;
        ws1_3.END TO sync3_4.END1;
        ws1_motors.RD_3 TO sync3_4.MOTOR1;
        ws1_motors.RD_4 TO sync3_4.MOTOR2;
        ws1_4.STYLO TO sync3_4.STYLE2;
        ws1_motors.RD_1 TO ws1_1.MTR_ON;
        ws1_4.END TO sync4_5.END1;
        ws1_motors.RD_4 TO sync4_5.MOTOR1;
        ws1_motors.RD_5 TO sync4_5.MOTOR2;
        ws1_5.STYLO TO sync4_5.STYLE2;
        ws1_1.END TO sync1_2.END1;
        ws1_motors.RD_1 TO sync1_2.MOTOR1;
        ws1_motors.RD_2 TO sync1_2.MOTOR2;
        ws1_2.STYLO TO sync1_2.STYLE2;
        ws1_motors.RD_2 TO sync2_3.MOTOR1;
        ws1_motors.RD_3 TO sync2_3.MOTOR2;
        ws1_3.STYLO TO sync2_3.STYLE2;
        ws1_2.END TO sync2_3.END1;
      END_CONNECTIONS
    END_RESOURCE
    RESOURCE WS3_model : PANEL_RESOURCE
      FBS
        ws3_1 : CNV_MDL(WKPC := [255,255,0], STYLE := VSTYLE#PALLET, VF := 10);
        ws3_2 : CNV_MDL(WKPC := [255,255,0], STYLE := VSTYLE#PALLET, VF := 10);
        ws3_3 : CNV_MDL(VF := 10, STYLE := VSTYLE#PALLET, WKPC := [255,255,0]);
        ws3_4 : CNV_MDL(VF := 10, STYLE := VSTYLE#PALLET, WKPC := [255,255,0]);
        ws3_5 : CNV_MDL(WKPC := [255,255,0], STYLE := VSTYLE#PALLET, VF := 10);
        ws3_pos : PUBL_5;
        ws3_sty : PUBL_5;
        ws3_motors : SUBL_5;
        ws3_op_load : SUBL_0;
        ws3_op_unload : SUBL_0;
        split5 : E_SPLIT;
        split4 : E_SPLIT;
        split3 : E_SPLIT;
        split2 : E_SPLIT;
        split1 : E_SPLIT;
        upd : SUBL_0;
        sync1_2 : ConvSync(STYLE1 := VSTYLE#NONE);
        sync2_3 : ConvSync(STYLE1 := VSTYLE#NONE);
        sync4_5 : ConvSync(STYLE1 := VSTYLE#NONE);
        sync3_4 : ConvSync(STYLE1 := VSTYLE#NONE);
      END_FBS
      EVENT_CONNECTIONS
        START.COLD TO ws3_motors.INIT;
        ws3_motors.INITO TO ws3_pos.INIT;
        ws3_pos.INITO TO ws3_sty.INIT;
        ws3_sty.INITO TO ws3_op_load.INIT;
        ws3_op_load.INITO TO ws3_op_unload.INIT;
        ws3_op_load.IND TO ws3_3.LOAD;
        ws3_op_unload.IND TO ws3_3.UNLD;
        ws3_pos.CNF TO ws3_sty.REQ;
        split1.EO2 TO split2.EI;
        split1.EO1 TO ws3_1.CLK;
        split2.EO2 TO split3.EI;
        split2.EO1 TO ws3_2.CLK;
        split3.EO2 TO split4.EI;
        split3.EO1 TO ws3_3.CLK;
        split4.EO2 TO split5.EI;
        split4.EO1 TO ws3_5.CLK;
        ws3_op_unload.INITO TO upd.INIT;
        upd.IND TO split1.EI;
        split5.EO2 TO ws3_pos.REQ;
        split5.EO1 TO ws3_4.CLK;
        sync3_4.CNF TO ws3_3.UNLD;
        sync3_4.CNF TO ws3_4.LOAD;
        split4.EO1 TO sync4_5.REQ;
        sync4_5.CNF TO ws3_4.UNLD;
        sync4_5.CNF TO ws3_5.LOAD;
        split3.EO1 TO sync3_4.REQ;
        split1.EO1 TO sync1_2.REQ;
        sync1_2.CNF TO ws3_2.LOAD;
        sync1_2.CNF TO ws3_1.UNLD;
        split2.EO1 TO sync2_3.REQ;
        sync2_3.CNF TO ws3_2.UNLD;
        sync2_3.CNF TO ws3_3.LOAD;
      END_CONNECTIONS
      DATA_CONNECTIONS
        ws3_1.POS TO ws3_pos.SD_1;
        ws3_2.POS TO ws3_pos.SD_2;
        ws3_3.POS TO ws3_pos.SD_3;
        ws3_4.POS TO ws3_pos.SD_4;
        ws3_5.POS TO ws3_pos.SD_5;
        ws3_1.STYLO TO ws3_sty.SD_1;
        ws3_2.STYLO TO ws3_sty.SD_2;
        ws3_3.STYLO TO ws3_sty.SD_3;
        ws3_4.STYLO TO ws3_sty.SD_4;
        ws3_5.STYLO TO ws3_sty.SD_5;
        ws3_motors.RD_2 TO ws3_2.MTR_ON;
        ws3_motors.RD_3 TO ws3_3.MTR_ON;
        ws3_motors.RD_4 TO ws3_4.MTR_ON;
        ws3_motors.RD_5 TO ws3_5.MTR_ON;
        ws3_3.END TO sync3_4.END1;
        ws3_motors.RD_3 TO sync3_4.MOTOR1;
        ws3_motors.RD_4 TO sync3_4.MOTOR2;
        ws3_4.STYLO TO sync3_4.STYLE2;
        ws3_motors.RD_1 TO ws3_1.MTR_ON;
        ws3_4.END TO sync4_5.END1;
        ws3_motors.RD_4 TO sync4_5.MOTOR1;
        ws3_motors.RD_5 TO sync4_5.MOTOR2;
        ws3_5.STYLO TO sync4_5.STYLE2;
        ws3_1.END TO sync1_2.END1;
        ws3_motors.RD_1 TO sync1_2.MOTOR1;
        ws3_motors.RD_2 TO sync1_2.MOTOR2;
        ws3_2.STYLO TO sync1_2.STYLE2;
        ws3_motors.RD_2 TO sync2_3.MOTOR1;
        ws3_motors.RD_3 TO sync2_3.MOTOR2;
        ws3_3.STYLO TO sync2_3.STYLE2;
        ws3_2.END TO sync2_3.END1;
      END_CONNECTIONS
    END_RESOURCE
    RESOURCE ML1_model : PANEL_RESOURCE
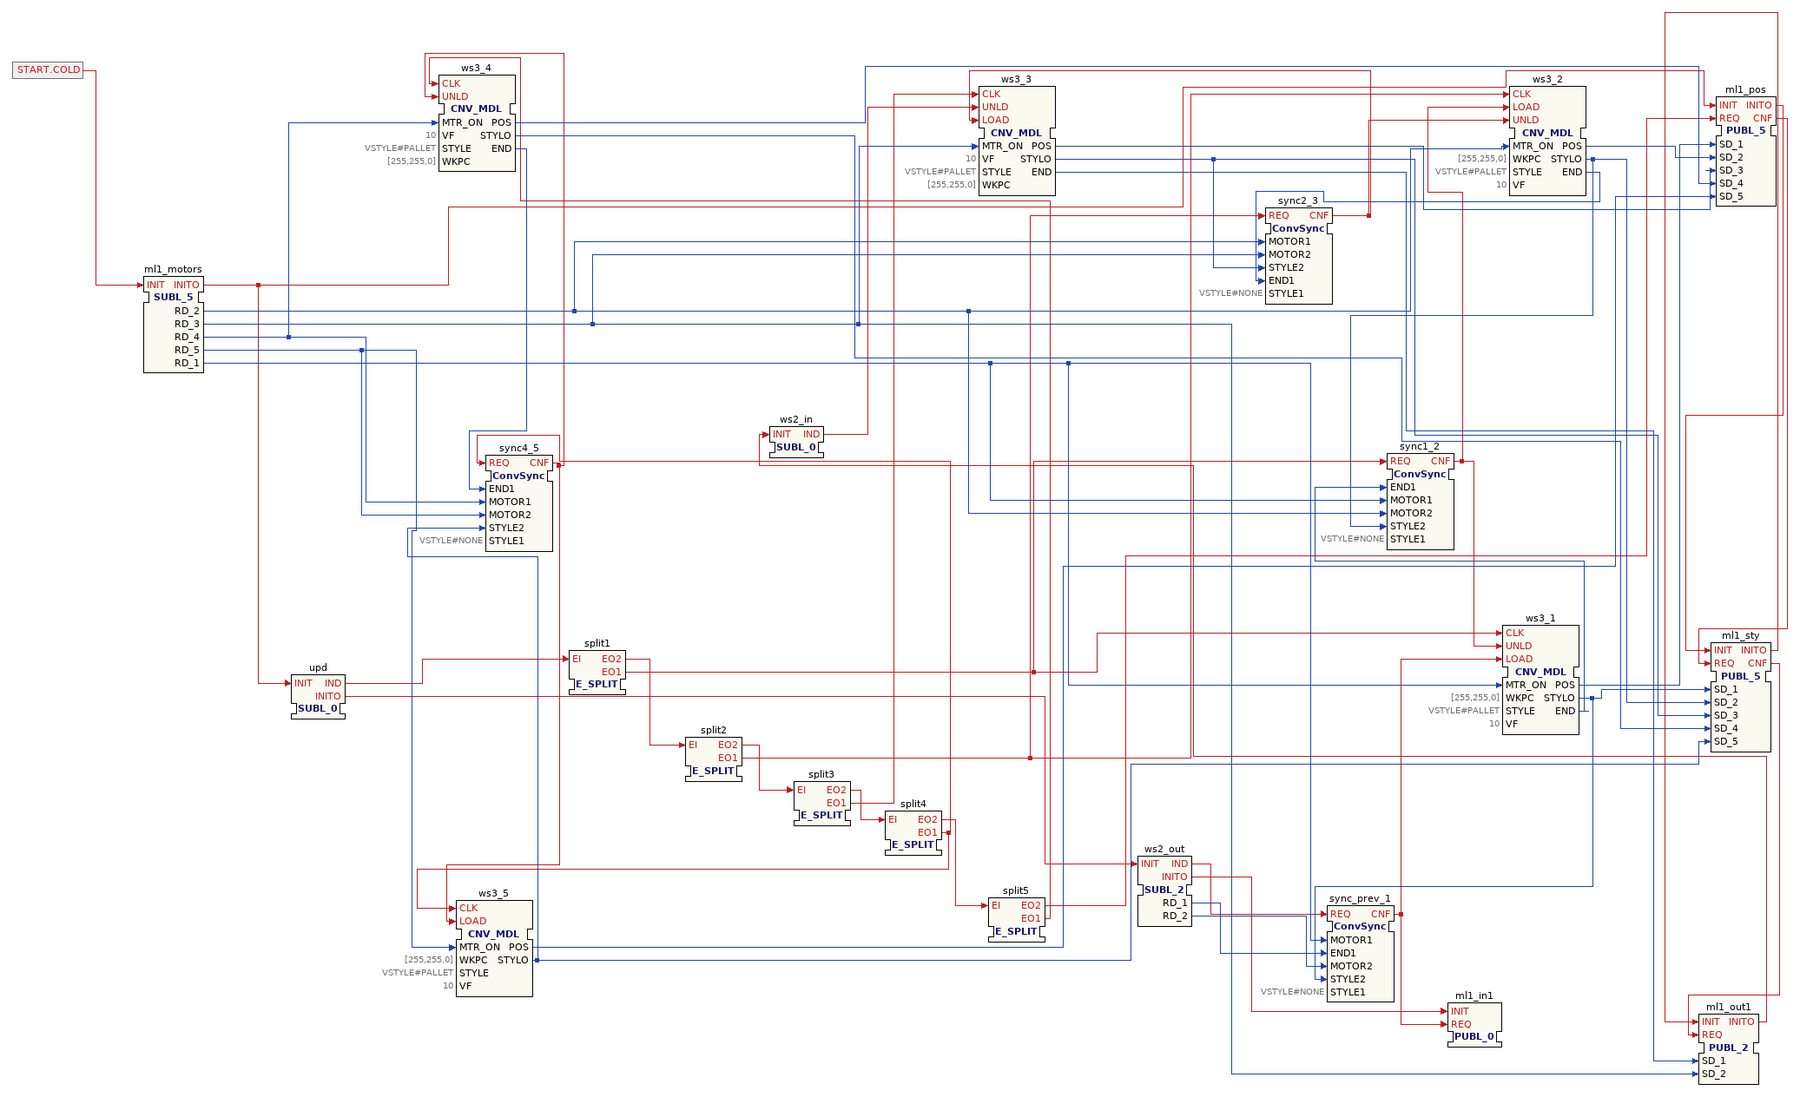
      FBS
        ws3_1 : CNV_MDL(WKPC := [255,255,0], STYLE := VSTYLE#PALLET, VF := 10);
        ws3_2 : CNV_MDL(WKPC := [255,255,0], STYLE := VSTYLE#PALLET, VF := 10);
        ws3_3 : CNV_MDL(VF := 10, STYLE := VSTYLE#PALLET, WKPC := [255,255,0]);
        ws3_4 : CNV_MDL(VF := 10, STYLE := VSTYLE#PALLET, WKPC := [255,255,0]);
        ws3_5 : CNV_MDL(WKPC := [255,255,0], STYLE := VSTYLE#PALLET, VF := 10);
        ml1_pos : PUBL_5;
        ml1_sty : PUBL_5;
        ml1_motors : SUBL_5;
        split5 : E_SPLIT;
        split4 : E_SPLIT;
        split3 : E_SPLIT;
        split2 : E_SPLIT;
        split1 : E_SPLIT;
        upd : SUBL_0;
        sync_prev_1 : ConvSync(STYLE1 := VSTYLE#NONE);
        sync1_2 : ConvSync(STYLE1 := VSTYLE#NONE);
        sync2_3 : ConvSync(STYLE1 := VSTYLE#NONE);
        sync4_5 : ConvSync(STYLE1 := VSTYLE#NONE);
        ml1_out1 : PUBL_2;
        ws2_in : SUBL_0;
        ws2_out : SUBL_2;
        ml1_in1 : PUBL_0;
      END_FBS
      EVENT_CONNECTIONS
        START.COLD TO ml1_motors.INIT;
        ml1_motors.INITO TO ml1_pos.INIT;
        ml1_pos.INITO TO ml1_sty.INIT;
        ml1_pos.CNF TO ml1_sty.REQ;
        split1.EO2 TO split2.EI;
        split1.EO1 TO ws3_1.CLK;
        split2.EO2 TO split3.EI;
        split2.EO1 TO ws3_2.CLK;
        split3.EO2 TO split4.EI;
        split3.EO1 TO ws3_3.CLK;
        split4.EO2 TO split5.EI;
        split4.EO1 TO ws3_5.CLK;
        upd.IND TO split1.EI;
        split5.EO2 TO ml1_pos.REQ;
        split5.EO1 TO ws3_4.CLK;
        split4.EO1 TO sync4_5.REQ;
        sync4_5.CNF TO ws3_4.UNLD;
        sync4_5.CNF TO ws3_5.LOAD;
        split1.EO1 TO sync1_2.REQ;
        sync1_2.CNF TO ws3_2.LOAD;
        sync1_2.CNF TO ws3_1.UNLD;
        split2.EO1 TO sync2_3.REQ;
        ml1_sty.INITO TO ml1_out1.INIT;
        ml1_sty.CNF TO ml1_out1.REQ;
        ws2_in.IND TO ws3_3.UNLD;
        sync2_3.CNF TO ws3_2.UNLD;
        sync2_3.CNF TO ws3_3.LOAD;
        ml1_out1.INITO TO ws2_in.INIT;
        ws2_out.IND TO sync_prev_1.REQ;
        ml1_motors.INITO TO upd.INIT;
        upd.INITO TO ws2_out.INIT;
        ws2_out.INITO TO ml1_in1.INIT;
        sync_prev_1.CNF TO ml1_in1.REQ;
        sync_prev_1.CNF TO ws3_1.LOAD;
      END_CONNECTIONS
      DATA_CONNECTIONS
        ws3_1.POS TO ml1_pos.SD_1;
        ws3_2.POS TO ml1_pos.SD_2;
        ws3_3.POS TO ml1_pos.SD_3;
        ws3_4.POS TO ml1_pos.SD_4;
        ws3_5.POS TO ml1_pos.SD_5;
        ws3_1.STYLO TO ml1_sty.SD_1;
        ws3_2.STYLO TO ml1_sty.SD_2;
        ws3_3.STYLO TO ml1_sty.SD_3;
        ws3_4.STYLO TO ml1_sty.SD_4;
        ws3_5.STYLO TO ml1_sty.SD_5;
        ml1_motors.RD_2 TO ws3_2.MTR_ON;
        ml1_motors.RD_3 TO ws3_3.MTR_ON;
        ml1_motors.RD_4 TO ws3_4.MTR_ON;
        ml1_motors.RD_5 TO ws3_5.MTR_ON;
        ml1_motors.RD_1 TO ws3_1.MTR_ON;
        ws3_4.END TO sync4_5.END1;
        ml1_motors.RD_4 TO sync4_5.MOTOR1;
        ml1_motors.RD_5 TO sync4_5.MOTOR2;
        ws3_5.STYLO TO sync4_5.STYLE2;
        ws3_1.END TO sync1_2.END1;
        ml1_motors.RD_1 TO sync1_2.MOTOR1;
        ml1_motors.RD_2 TO sync1_2.MOTOR2;
        ws3_2.STYLO TO sync1_2.STYLE2;
        ml1_motors.RD_2 TO sync2_3.MOTOR1;
        ml1_motors.RD_3 TO sync2_3.MOTOR2;
        ws3_3.STYLO TO sync2_3.STYLE2;
        ws3_2.END TO sync2_3.END1;
        ml1_motors.RD_1 TO sync_prev_1.MOTOR1;
        ws2_out.RD_1 TO sync_prev_1.END1;
        ws2_out.RD_2 TO sync_prev_1.MOTOR2;
        ws3_1.STYLO TO sync_prev_1.STYLE2;
        ws3_3.END TO ml1_out1.SD_1;
        ml1_motors.RD_3 TO ml1_out1.SD_2;
      END_CONNECTIONS
    END_RESOURCE
  END_DEVICE
  DEVICE View : FRAME_DEVICE(BOUNDS := [200,450,720,360])
    RESOURCE Canvas : VIEW_PANEL(DIA := 20, SIZE := [36,16])
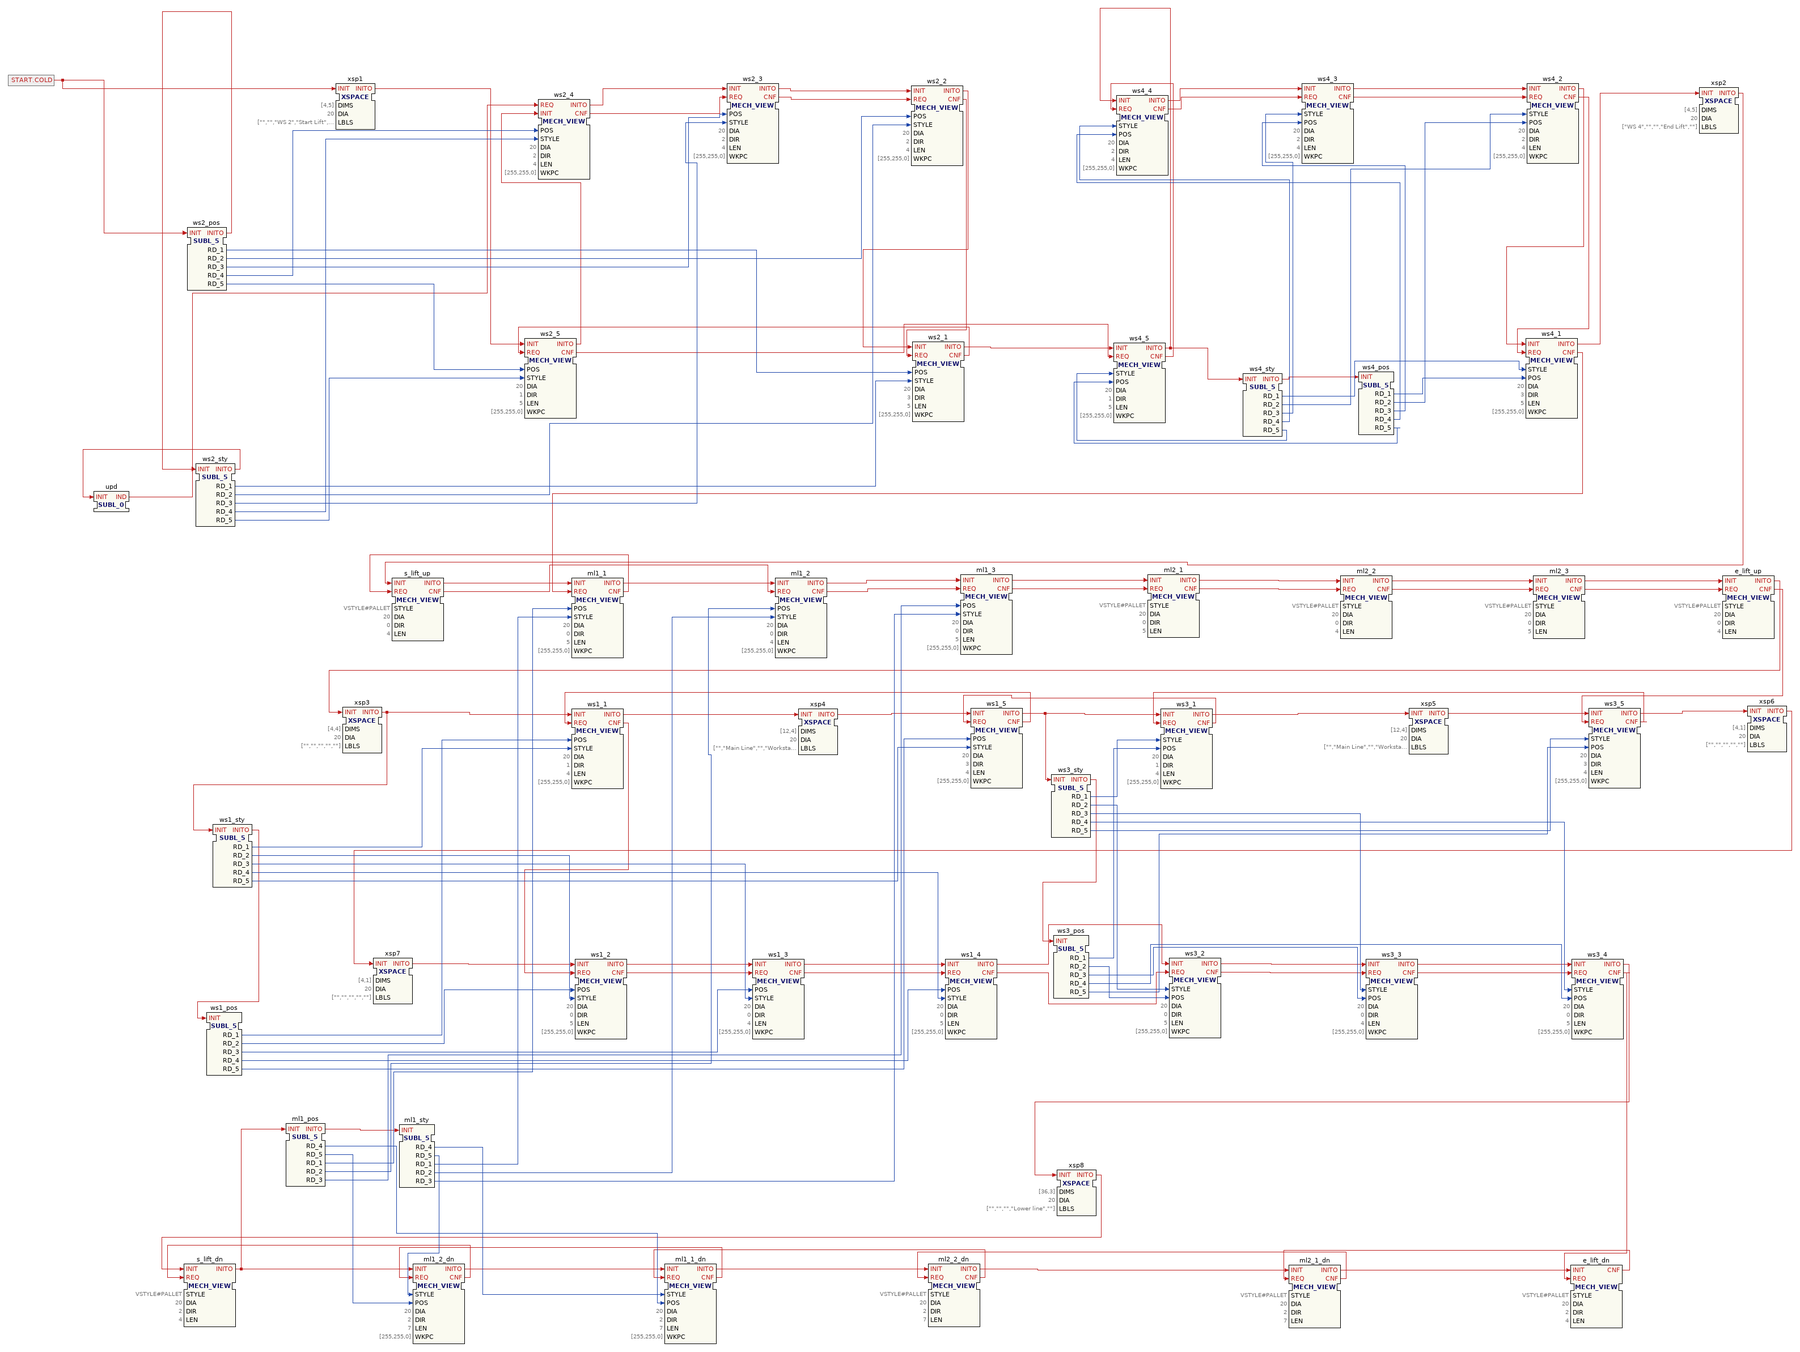
      FBS
        xsp1 : XSPACE(DIMS := [4,5], DIA := 20, LBLS := ["","","WS 2","Start Lift",""]);
        xsp3 : XSPACE(DIMS := [4,4], DIA := 20, LBLS := ["","","","",""]);
        ws2_4 : MECH_VIEW(DIA := 20, DIR := 2, LEN := 4, WKPC := [255,255,0]);
        ws2_3 : MECH_VIEW(DIA := 20, DIR := 2, LEN := 4, WKPC := [255,255,0]);
        ws2_2 : MECH_VIEW(DIA := 20, DIR := 2, LEN := 4, WKPC := [255,255,0]);
        ws4_4 : MECH_VIEW(DIA := 20, DIR := 2, LEN := 4, WKPC := [255,255,0]);
        ws4_3 : MECH_VIEW(DIA := 20, DIR := 2, LEN := 4, WKPC := [255,255,0]);
        ws4_2 : MECH_VIEW(DIA := 20, DIR := 2, LEN := 4, WKPC := [255,255,0]);
        ws2_5 : MECH_VIEW(DIA := 20, DIR := 1, LEN := 5, WKPC := [255,255,0]);
        s_lift_up : MECH_VIEW(STYLE := VSTYLE#PALLET, DIA := 20, DIR := 0, LEN := 4);
        ml1_1 : MECH_VIEW(DIA := 20, DIR := 0, LEN := 5, WKPC := [255,255,0]);
        ml1_2 : MECH_VIEW(DIA := 20, DIR := 0, LEN := 4, WKPC := [255,255,0]);
        ml1_3 : MECH_VIEW(DIA := 20, DIR := 0, LEN := 5, WKPC := [255,255,0]);
        ml2_1 : MECH_VIEW(STYLE := VSTYLE#PALLET, DIA := 20, DIR := 0, LEN := 5);
        ml2_2 : MECH_VIEW(STYLE := VSTYLE#PALLET, DIA := 20, DIR := 0, LEN := 4);
        ml2_3 : MECH_VIEW(STYLE := VSTYLE#PALLET, DIA := 20, DIR := 0, LEN := 5);
        e_lift_up : MECH_VIEW(STYLE := VSTYLE#PALLET, DIA := 20, DIR := 0, LEN := 4);
        ws2_1 : MECH_VIEW(DIA := 20, DIR := 3, LEN := 5, WKPC := [255,255,0]);
        ws4_5 : MECH_VIEW(DIA := 20, DIR := 1, LEN := 5, WKPC := [255,255,0]);
        ws4_1 : MECH_VIEW(DIA := 20, DIR := 3, LEN := 5, WKPC := [255,255,0]);
        xsp2 : XSPACE(DIMS := [4,5], DIA := 20, LBLS := ["WS 4","","","End Lift",""]);
        ws1_1 : MECH_VIEW(DIA := 20, DIR := 1, LEN := 4, WKPC := [255,255,0]);
        ws1_2 : MECH_VIEW(DIA := 20, DIR := 0, LEN := 5, WKPC := [255,255,0]);
        ws1_3 : MECH_VIEW(DIA := 20, DIR := 0, LEN := 4, WKPC := [255,255,0]);
        ws1_4 : MECH_VIEW(DIA := 20, DIR := 0, LEN := 5, WKPC := [255,255,0]);
        ws1_5 : MECH_VIEW(DIA := 20, DIR := 3, LEN := 4, WKPC := [255,255,0]);
        ws3_1 : MECH_VIEW(DIA := 20, DIR := 1, LEN := 4, WKPC := [255,255,0]);
        ws3_2 : MECH_VIEW(DIA := 20, DIR := 0, LEN := 5, WKPC := [255,255,0]);
        ws3_3 : MECH_VIEW(DIA := 20, DIR := 0, LEN := 4, WKPC := [255,255,0]);
        ws3_4 : MECH_VIEW(DIA := 20, DIR := 0, LEN := 5, WKPC := [255,255,0]);
        ws3_5 : MECH_VIEW(DIA := 20, DIR := 3, LEN := 4, WKPC := [255,255,0]);
        xsp4 : XSPACE(DIMS := [12,4], DIA := 20, LBLS := ["","Main Line","","Workstation 1",""]);
        xsp5 : XSPACE(DIMS := [12,4], DIA := 20, LBLS := ["","Main Line","","Workstation 3",""]);
        xsp6 : XSPACE(DIMS := [4,1], DIA := 20, LBLS := ["","","","",""]);
        xsp7 : XSPACE(DIMS := [4,1], DIA := 20, LBLS := ["","","","",""]);
        xsp8 : XSPACE(DIMS := [36,3], DIA := 20, LBLS := ["","","","Lower line",""]);
        s_lift_dn : MECH_VIEW(STYLE := VSTYLE#PALLET, DIA := 20, DIR := 2, LEN := 4);
        ml1_1_dn : MECH_VIEW(DIA := 20, DIR := 2, LEN := 7, WKPC := [255,255,0]);
        ml1_2_dn : MECH_VIEW(DIA := 20, DIR := 2, LEN := 7, WKPC := [255,255,0]);
        ml2_1_dn : MECH_VIEW(STYLE := VSTYLE#PALLET, DIA := 20, DIR := 2, LEN := 7);
        ml2_2_dn : MECH_VIEW(STYLE := VSTYLE#PALLET, DIA := 20, DIR := 2, LEN := 7);
        e_lift_dn : MECH_VIEW(STYLE := VSTYLE#PALLET, DIA := 20, DIR := 2, LEN := 4);
        ws4_pos : SUBL_5;
        ws3_pos : SUBL_5;
        ml1_pos : SUBL_5;
        ws1_pos : SUBL_5;
        ws2_pos : SUBL_5;
        ws4_sty : SUBL_5;
        ws3_sty : SUBL_5;
        ml1_sty : SUBL_5;
        ws1_sty : SUBL_5;
        ws2_sty : SUBL_5;
        upd : SUBL_0;
      END_FBS
      EVENT_CONNECTIONS
        START.COLD TO xsp1.INIT;
        ws2_3.INITO TO ws2_2.INIT;
        ws4_4.INITO TO ws4_3.INIT;
        ws4_3.INITO TO ws4_2.INIT;
        xsp1.INITO TO ws2_5.INIT;
        ws2_4.INITO TO ws2_3.INIT;
        ws2_2.INITO TO ws2_1.INIT;
        ws2_1.INITO TO ws4_5.INIT;
        ws4_5.INITO TO ws4_4.INIT;
        ws4_2.INITO TO ws4_1.INIT;
        ws4_1.INITO TO xsp2.INIT;
        xsp2.INITO TO s_lift_up.INIT;
        s_lift_up.INITO TO ml1_1.INIT;
        ml1_1.INITO TO ml1_2.INIT;
        ml1_2.INITO TO ml1_3.INIT;
        ml1_3.INITO TO ml2_1.INIT;
        ml2_1.INITO TO ml2_2.INIT;
        ml2_2.INITO TO ml2_3.INIT;
        ml2_3.INITO TO e_lift_up.INIT;
        e_lift_up.INITO TO xsp3.INIT;
        xsp3.INITO TO ws1_1.INIT;
        ws1_2.INITO TO ws1_3.INIT;
        ws1_3.INITO TO ws1_4.INIT;
        ws3_2.INITO TO ws3_3.INIT;
        ws3_3.INITO TO ws3_4.INIT;
        ws1_1.INITO TO xsp4.INIT;
        xsp4.INITO TO ws1_5.INIT;
        ws1_5.INITO TO ws3_1.INIT;
        ws3_1.INITO TO xsp5.INIT;
        xsp5.INITO TO ws3_5.INIT;
        ws1_4.INITO TO ws3_2.INIT;
        xsp7.INITO TO ws1_2.INIT;
        ws3_5.INITO TO xsp6.INIT;
        xsp6.INITO TO xsp7.INIT;
        ws3_4.INITO TO xsp8.INIT;
        ml2_1_dn.INITO TO e_lift_dn.INIT;
        ml2_2_dn.INITO TO ml2_1_dn.INIT;
        ml1_1_dn.INITO TO ml2_2_dn.INIT;
        ml1_2_dn.INITO TO ml1_1_dn.INIT;
        s_lift_dn.INITO TO ml1_2_dn.INIT;
        xsp8.INITO TO s_lift_dn.INIT;
        START.COLD TO ws2_pos.INIT;
        ws2_pos.INITO TO ws2_sty.INIT;
        ws2_4.CNF TO ws2_3.REQ;
        ws2_3.CNF TO ws2_2.REQ;
        ws2_2.CNF TO ws2_1.REQ;
        ws2_1.CNF TO ws2_5.REQ;
        upd.IND TO ws2_4.REQ;
        ws2_sty.INITO TO upd.INIT;
        ws4_4.CNF TO ws4_3.REQ;
        ws2_5.INITO TO ws2_4.INIT;
        ws2_5.CNF TO ws4_5.REQ;
        ws4_5.CNF TO ws4_4.REQ;
        ws4_3.CNF TO ws4_2.REQ;
        ws4_2.CNF TO ws4_1.REQ;
        ws4_sty.INITO TO ws4_pos.INIT;
        ws4_5.INITO TO ws4_sty.INIT;
        ws4_1.CNF TO ml1_1.REQ;
        ml1_1.CNF TO s_lift_up.REQ;
        s_lift_up.CNF TO ml1_2.REQ;
        ml1_2.CNF TO ml1_3.REQ;
        ml1_3.CNF TO ml2_1.REQ;
        ml2_1.CNF TO ml2_2.REQ;
        ml2_2.CNF TO ml2_3.REQ;
        ml2_3.CNF TO e_lift_up.REQ;
        e_lift_up.CNF TO ws3_5.REQ;
        ws3_5.CNF TO ws3_1.REQ;
        ws3_1.CNF TO ws1_5.REQ;
        ws1_5.CNF TO ws1_1.REQ;
        ws1_1.CNF TO ws1_2.REQ;
        ws1_2.CNF TO ws1_3.REQ;
        ws1_3.CNF TO ws1_4.REQ;
        ws1_4.CNF TO ws3_2.REQ;
        ws3_2.CNF TO ws3_3.REQ;
        ws3_3.CNF TO ws3_4.REQ;
        ws3_4.CNF TO e_lift_dn.REQ;
        e_lift_dn.CNF TO ml2_1_dn.REQ;
        ml2_1_dn.CNF TO ml2_2_dn.REQ;
        ml2_2_dn.CNF TO ml1_1_dn.REQ;
        ml1_1_dn.CNF TO ml1_2_dn.REQ;
        ml1_2_dn.CNF TO s_lift_dn.REQ;
        xsp3.INITO TO ws1_sty.INIT;
        ws1_sty.INITO TO ws1_pos.INIT;
        ws1_5.INITO TO ws3_sty.INIT;
        ws3_sty.INITO TO ws3_pos.INIT;
        s_lift_dn.INITO TO ml1_pos.INIT;
        ml1_pos.INITO TO ml1_sty.INIT;
      END_CONNECTIONS
      DATA_CONNECTIONS
        ws2_pos.RD_1 TO ws2_1.POS;
        ws2_pos.RD_2 TO ws2_2.POS;
        ws2_pos.RD_3 TO ws2_3.POS;
        ws2_pos.RD_4 TO ws2_4.POS;
        ws2_pos.RD_5 TO ws2_5.POS;
        ws2_sty.RD_1 TO ws2_1.STYLE;
        ws2_sty.RD_2 TO ws2_2.STYLE;
        ws2_sty.RD_3 TO ws2_3.STYLE;
        ws2_sty.RD_4 TO ws2_4.STYLE;
        ws2_sty.RD_5 TO ws2_5.STYLE;
        ws4_sty.RD_1 TO ws4_1.STYLE;
        ws4_sty.RD_2 TO ws4_2.STYLE;
        ws4_sty.RD_3 TO ws4_3.STYLE;
        ws4_sty.RD_4 TO ws4_4.STYLE;
        ws4_sty.RD_5 TO ws4_5.STYLE;
        ws4_pos.RD_1 TO ws4_1.POS;
        ws4_pos.RD_2 TO ws4_2.POS;
        ws4_pos.RD_3 TO ws4_3.POS;
        ws4_pos.RD_4 TO ws4_4.POS;
        ws4_pos.RD_5 TO ws4_5.POS;
        ws1_pos.RD_1 TO ws1_1.POS;
        ws1_pos.RD_2 TO ws1_2.POS;
        ws1_pos.RD_3 TO ws1_3.POS;
        ws1_pos.RD_4 TO ws1_4.POS;
        ws1_pos.RD_5 TO ws1_5.POS;
        ws1_sty.RD_1 TO ws1_1.STYLE;
        ws1_sty.RD_2 TO ws1_2.STYLE;
        ws1_sty.RD_3 TO ws1_3.STYLE;
        ws1_sty.RD_4 TO ws1_4.STYLE;
        ws1_sty.RD_5 TO ws1_5.STYLE;
        ws3_sty.RD_1 TO ws3_1.STYLE;
        ws3_sty.RD_2 TO ws3_2.STYLE;
        ws3_sty.RD_3 TO ws3_3.STYLE;
        ws3_sty.RD_4 TO ws3_4.STYLE;
        ws3_sty.RD_5 TO ws3_5.STYLE;
        ws3_pos.RD_1 TO ws3_1.POS;
        ws3_pos.RD_2 TO ws3_2.POS;
        ws3_pos.RD_3 TO ws3_3.POS;
        ws3_pos.RD_4 TO ws3_4.POS;
        ws3_pos.RD_5 TO ws3_5.POS;
        ml1_sty.RD_4 TO ml1_1_dn.STYLE;
        ml1_sty.RD_5 TO ml1_2_dn.STYLE;
        ml1_pos.RD_4 TO ml1_1_dn.POS;
        ml1_pos.RD_5 TO ml1_2_dn.POS;
        ml1_pos.RD_1 TO ml1_1.POS;
        ml1_pos.RD_2 TO ml1_2.POS;
        ml1_pos.RD_3 TO ml1_3.POS;
        ml1_sty.RD_1 TO ml1_1.STYLE;
        ml1_sty.RD_2 TO ml1_2.STYLE;
        ml1_sty.RD_3 TO ml1_3.STYLE;
      END_CONNECTIONS
    END_RESOURCE
  END_DEVICE
END_SYSTEM
